TYPE "EFC_CONTROL_WORD"
VERSION : 0.1
// Block: EFC_CONTROL_WORD
   STRUCT
      FreeWheelingStop : Bool;
      TorqueControl : Bool;
      Reserved2 : Bool;
      Reserved3 : Bool;
      Reserved4 : Bool;
      Reserved5 : Bool;
      Reserved6 : Bool;
      Reserved7 : Bool;
      Run : Bool;
      Jog : Bool;
      Reverse : Bool;
      StopParameter : Bool;
      EStop : Bool;
      ErrorReset : Bool;
      StopAccDec : Bool;
      ControlWord : Bool;
   END_STRUCT;

END_TYPE
